// TIA Portal V20 export
DATA_BLOCK "Instance Machine Modules"   // DB1
// stored: InstanceOfName FB - Machine Modules, InstanceOfType FB
"FB - Machine Modules"
BEGIN
END_DATA_BLOCK
